(* CoDeSys 2.3.9.41 project: hlor-rezerv.pro *)
(* Libraries: STANDARD.LIB 4.10.05 11:14:46, IECSFC.LIB 13.4.06 15:51:28, ANALYZATION.LIB 5.10.99 09:05:06 *)

(* PLC configuration (modules and I/O channels)
Fast discrete inputs [I_SIMPLE_INPUT] node 0, in %IB0 out %QB0 {ChannellName = Fast discrete inputs; Filtrationtime = 10000}
  AT %IX0.0 [BitInput] Discrete input 1 {ChannellName = Enter name}
  AT %IX0.1 [BitInput] Discrete input 2 {ChannellName = Enter name}
  AT %IX0.2 [BitInput] Discrete input 3 {ChannellName = Enter name}
  AT %IX0.3 [BitInput] Discrete input 4 {ChannellName = Enter name}
Discrete inputs [ID130] node 1, in %IB1 out %QB1 {ChannellName = Discrete inputs; Filtrationtime_GeneralINP = 10; PinCount = 12; Visibility = No}
  AT %IB1.0 [ByteInput] 8 discrete inputs {ChannellName = Enter name}
  AT %IB1.1 [ByteInput] 4 discrete inputs {ChannellName = Enter name}
Fast discrete outputs [OWEN_ID570] node 2, in %IB2 out %QB2 {ChannellName = Fast discrete outputs; SafeValueBool = FALSE; SafeValueBool = FALSE; SafeValueBool = FALSE; SafeValueBool = FALSE; Visibility = No}
  SolNasos AT %QX2.0 [BitOutput] Fast discrete output 1 {ChannellName = Enter name}
  WaterNasos AT %QX2.1 [BitOutput] Fast discrete output 2 {ChannellName = Enter name}
  Klapan AT %QX2.2 [BitOutput] Fast discrete output 3 {ChannellName = Enter name}
  Elektroliz AT %QX2.3 [BitOutput] Fast discrete output 4 {ChannellName = Enter name}
Discrete outputs [ID131] node 3, in %IB3 out %QB3 {ChannellName = Discrete outputs; SafeValueByte = 0; Visibility = No}
  AT %QB3.0 [ByteOutput] 8 discrete outputs {ChannellName = Enter name}
  AT %QB3.1 [ByteOutput] 8 discrete outputs {ChannellName = Enter name}
D_Volume_Bak AT %IR4.0 [FloatInputP] Объем бака {ChannellName = Fast analog input; AIN_TYPE = 4-20 mA; Peak_Filtr = 200; Flt_Ch = Off; TauRC = 10; MinFV = 0; MaxFV = 150}
D_Konduktivnost AT %IR4.1 [FloatInputP] D_Konduktivnost {ChannellName = Fast analog input; AIN_TYPE = 4-20 mA; Peak_Filtr = 200; Flt_Ch = Off; TauRC = 10; MinFV = 0; MaxFV = 200}
D_Volt AT %IR4.2 [FloatInputP] Ток выпрямителя {ChannellName = Fast analog input; AIN_TYPE = 4-20 mA; Peak_Filtr = 200; Flt_Ch = Off; TauRC = 10; MinFV = 0; MaxFV = 80}
D_Amper AT %IR4.3 [FloatInputP] Напряжение выпрямителя {ChannellName = Fast analog input; AIN_TYPE = 4-20 mA; Peak_Filtr = 200; Flt_Ch = Off; TauRC = 10; MinFV = 0; MaxFV = 200}
DT_Water_Input AT %IR4.4 [FloatInputP] Температура воды на входе {ChannellName = Fast analog input; AIN_TYPE = 4-20 mA; Peak_Filtr = 200; Flt_Ch = Off; TauRC = 10; MinFV = 0; MaxFV = 100}
DT_Water_output AT %IR4.5 [FloatInputP] Температура воды на выходе {ChannellName = Fast analog input; AIN_TYPE = 4-20 mA; Peak_Filtr = 200; Flt_Ch = Off; TauRC = 10; MinFV = 0; MaxFV = 100}
AT %IR4.6 [FloatInputP] {ChannellName = Fast analog input; AIN_TYPE = 4-20 mA; Peak_Filtr = 200; Flt_Ch = Off; TauRC = 10; MinFV = 0; MaxFV = 100}
AT %IR4.7 [FloatInputP] You need to reboot PLC after change AI configuration! {ChannellName = Fast analog input; AIN_TYPE = 4-20 mA; Peak_Filtr = 200; Flt_Ch = Off; TauRC = 10; MinFV = 0; MaxFV = 20000.0}
AT %IW4.8 [WordInput] AI read time (10ms) {ChannellName = Enter name}
Analog outputs [ID126] node 5, in %IB5 out %QB5 {ChannellName = Analog outputs}
  AT %QR5.0 [FloatOutputP] AO #1 {ChannellName = Analog output; AOUT_TYPE = 4-20 mA; SafeValueREAL = 0.0}
  AT %QR5.1 [FloatOutputP] AO #2 {ChannellName = Analog output; AOUT_TYPE = 4-20 mA; SafeValueREAL = 0.0}
  AT %QR5.2 [FloatOutputP] AO #3 {ChannellName = Analog output; AOUT_TYPE = 4-20 mA; SafeValueREAL = 0.0}
  AT %QR5.3 [FloatOutputP] AO #4 {ChannellName = Analog output; AOUT_TYPE = 4-20 mA; SafeValueREAL = 0.0}
Special input [ID103] node 6, in %IB6 out %QB6 {ChannellName = Special input}
  AT %IX6.0 [BitInput] Special input {ChannellName = Enter name}
Special output [ID104] node 7, in %IB7 out %QB7 {ChannellName = Special output}
  AT %QX7.0 [BitOutput] Special output {ChannellName = Enter name}
Modbus [MODBUS_ID302] node 0, in %IB8.0 out %QB8.0 {ChannellName = Modbus}
  TCP [TCP_ID221] node 0, in %IB8.0.0 out %QB8.0.0 {ChannellName = TCP; RemotePort = 502; Visibility = No}
8 bits [8Bit] node 1, in %IB8.1 out %QB8.1 {ChannellName = 8 bit}
  AT %QB8.1.0 [ByteOutput] {ChannellName = Enter name}
8 bits [8Bit] node 2, in %IB8.2 out %QB8.2 {ChannellName = 8 bit}
  AT %QB8.2.0 [ByteOutput] {ChannellName = Enter name}
8 bits [8Bit] node 3, in %IB8.3 out %QB8.3 {ChannellName = 8 bit}
  AT %QB8.3.0 [ByteOutput] {ChannellName = Enter name}
8 bits [8Bit] node 4, in %IB8.4 out %QB8.4 {ChannellName = 8 bit}
  AT %QB8.4.0 [ByteOutput] {ChannellName = Enter name}
8 bits [8Bit] node 5, in %IB8.5 out %QB8.5 {ChannellName = 8 bit}
  AT %QB8.5.0 [ByteOutput] {ChannellName = Enter name}
8 bits [8Bit] node 6, in %IB8.6 out %QB8.6 {ChannellName = 8 bit}
  AT %QB8.6.0 [ByteOutput] {ChannellName = Enter name}
Float [Float] node 7, in %IB8.7 out %QB8.7 {ChannellName = float}
  D_Volume_Bak_SPK AT %QD8.7.0 [FloatOutput] {ChannellName = Enter name}
Float [Float] node 8, in %IB8.8 out %QB8.8 {ChannellName = float}
  D_Konduktivnost_SPK AT %QD8.8.0 [FloatOutput] {ChannellName = Enter name}
  D_Volt_SPK AT %QD8.9.0 [FloatOutput] {ChannellName = Enter name}
  D_Amper_SPK AT %QD8.10.0 [FloatOutput] {ChannellName = Enter name}
Float [Float] node 11, in %IB8.11 out %QB8.11 {ChannellName = float}
  DT_Water_Input_SPK AT %QD8.11.0 [FloatOutput] {ChannellName = Enter name}
Float [Float] node 12, in %IB8.12 out %QB8.12 {ChannellName = float}
  DT_Water_output_SPK AT %QD8.12.0 [FloatOutput] {ChannellName = Enter name}
8 bits [8Bit] node 13, in %IB8.13 out %QB8.13 {ChannellName = 8 bit}
  AT %QB8.13.0 [ByteOutput] {ChannellName = Enter name}
8 bits [8Bit] node 14, in %IB8.14 out %QB8.14 {ChannellName = 8 bit}
  AT %QB8.14.0 [ByteOutput] {ChannellName = Enter name}
8 bits [8Bit] node 15, in %IB8.15 out %QB8.15 {ChannellName = 8 bit}
  AT %QB8.15.0 [ByteOutput] {ChannellName = Enter name}
8 bits [8Bit] node 16, in %IB8.16 out %QB8.16 {ChannellName = 8 bit}
  AT %QB8.16.0 [ByteOutput] {ChannellName = Enter name}
*)

(* Task configuration *)
TASK NewTask (PRIORITY := 1, INTERVAL := T#200ms);
	PLC_PRG();
END_TASK

(* Global variable list: Global_Variables *)
VAR_GLOBAL
	PLAY_Elektroliz: BOOL;
	StartElectroliz: BOOL;
	StopElectroliz: BOOL;
	StartKlap: BOOL;
	StoptKlap: BOOL;
	StartWaterNasos: BOOL;
	StopWaterNasos: BOOL;
	StartSolNasos: BOOL;
	StopSolNasos: BOOL;
	StartHlorNasos1: BOOL;
	StopHlorNasos1: BOOL;
	StartHlorNasos2: BOOL;
	StopHlorNasos2: BOOL;

	StartVozduh: BOOL;
	StopVozduh: BOOL;
END_VAR

(* POU PLC_PRG, CFC *)
(*
	Программа управления гипохлоридной установкой
	Контроллер ОВЕН ПЛК-160 M2
	Панель оператора Kinko MT4404T

*)


PROGRAM PLC_PRG
VAR
	Electroliz_prg: Electroliz;
	Hlorirovanie_prg: Hlorirovanie;
	SoftWater_prg: SoftWater;
	SolNasos_prg: SolNasos;
	Vozduh_prg: Vozduh;
	D_Elektroliz_prg: D_Elektroliz;
END_VAR
VAR (* helpers for the ST form of the networks *)
	_t97 : WORD;
	_t98 : WORD;
	_t99 : WORD;
	_t100 : WORD;
	_t101 : WORD;
	_t204 : WORD;
END_VAR
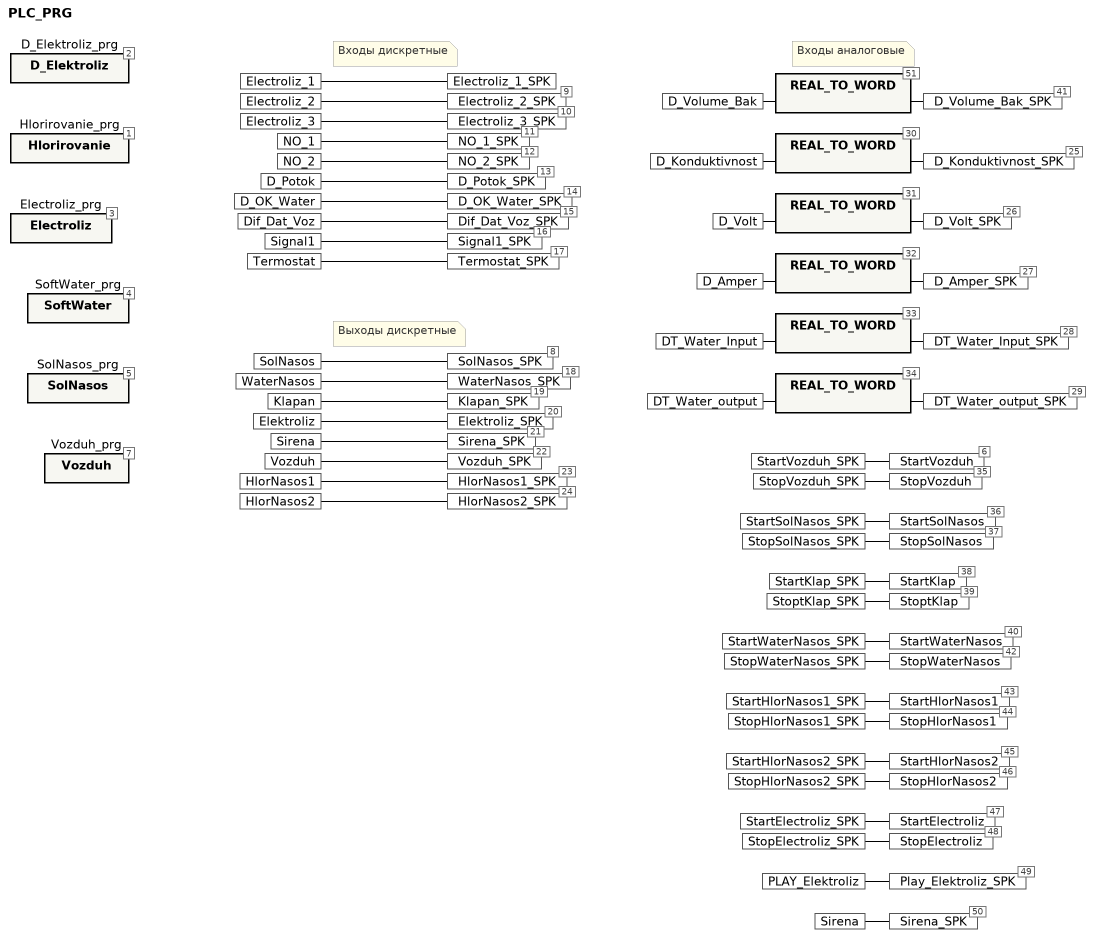
_CFC_ (* Continuous Function Chart, elements in execution order *)
#0 Electroliz_1_SPK <= Electroliz_1
#1 Hlorirovanie_prg:Hlorirovanie()
(* Входы дискретные *)
#2 D_Elektroliz_prg:D_Elektroliz()
#3 Electroliz_prg:Electroliz()
#4 SoftWater_prg:SoftWater()
#5 SolNasos_prg:SolNasos()
#6 StartVozduh <= StartVozduh_SPK
#7 Vozduh_prg:Vozduh()
(* Выходы дискретные *)
#8 SolNasos_SPK <= SolNasos
#9 Electroliz_2_SPK <= Electroliz_2
#10 Electroliz_3_SPK <= Electroliz_3
#11 NO_1_SPK <= NO_1
#12 NO_2_SPK <= NO_2
#13 D_Potok_SPK <= D_Potok
#14 D_OK_Water_SPK <= D_OK_Water
#15 Dif_Dat_Voz_SPK <= Dif_Dat_Voz
#16 Signal1_SPK <= Signal1
#17 Termostat_SPK <= Termostat
#18 WaterNasos_SPK <= WaterNasos
#19 Klapan_SPK <= Klapan
#20 Elektroliz_SPK <= Elektroliz
#21 Sirena_SPK <= Sirena
#22 Vozduh_SPK <= Vozduh
#23 HlorNasos1_SPK <= HlorNasos1
#24 HlorNasos2_SPK <= HlorNasos2
(* Входы аналоговые *)
#25 D_Konduktivnost_SPK <= #30
#26 D_Volt_SPK <= #31
#27 D_Amper_SPK <= #32
#28 DT_Water_Input_SPK <= #33
#29 DT_Water_output_SPK <= #34
#30 REAL_TO_WORD(D_Konduktivnost)
#31 REAL_TO_WORD(D_Volt)
#32 REAL_TO_WORD(D_Amper)
#33 REAL_TO_WORD(DT_Water_Input)
#34 REAL_TO_WORD(DT_Water_output)
#35 StopVozduh <= StopVozduh_SPK
#36 StartSolNasos <= StartSolNasos_SPK
#37 StopSolNasos <= StopSolNasos_SPK
#38 StartKlap <= StartKlap_SPK
#39 StoptKlap <= StoptKlap_SPK
#40 StartWaterNasos <= StartWaterNasos_SPK
#41 D_Volume_Bak_SPK <= #51
#42 StopWaterNasos <= StopWaterNasos_SPK
#43 StartHlorNasos1 <= StartHlorNasos1_SPK
#44 StopHlorNasos1 <= StopHlorNasos1_SPK
#45 StartHlorNasos2 <= StartHlorNasos2_SPK
#46 StopHlorNasos2 <= StopHlorNasos2_SPK
#47 StartElectroliz <= StartElectroliz_SPK
#48 StopElectroliz <= StopElectroliz_SPK
#49 Play_Elektroliz_SPK <= PLAY_Elektroliz
#50 Sirena_SPK <= Sirena
#51 REAL_TO_WORD(D_Volume_Bak)
_END_CFC_
(* the same logic as Structured Text *)
Electroliz_1_SPK := Electroliz_1;
Hlorirovanie_prg();
(* Входы дискретные *)
D_Elektroliz_prg();
Electroliz_prg();
SoftWater_prg();
SolNasos_prg();
StartVozduh := StartVozduh_SPK;
Vozduh_prg();
(* Выходы дискретные *)
SolNasos_SPK := SolNasos;
Electroliz_2_SPK := Electroliz_2;
Electroliz_3_SPK := Electroliz_3;
NO_1_SPK := NO_1;
NO_2_SPK := NO_2;
D_Potok_SPK := D_Potok;
D_OK_Water_SPK := D_OK_Water;
Dif_Dat_Voz_SPK := Dif_Dat_Voz;
Signal1_SPK := Signal1;
Termostat_SPK := Termostat;
WaterNasos_SPK := WaterNasos;
Klapan_SPK := Klapan;
Elektroliz_SPK := Elektroliz;
Sirena_SPK := Sirena;
Vozduh_SPK := Vozduh;
HlorNasos1_SPK := HlorNasos1;
HlorNasos2_SPK := HlorNasos2;
(* Входы аналоговые *)
D_Konduktivnost_SPK := _t97;
D_Volt_SPK := _t98;
D_Amper_SPK := _t99;
DT_Water_Input_SPK := _t100;
DT_Water_output_SPK := _t101;
_t97 := REAL_TO_WORD(D_Konduktivnost);
_t98 := REAL_TO_WORD(D_Volt);
_t99 := REAL_TO_WORD(D_Amper);
_t100 := REAL_TO_WORD(DT_Water_Input);
_t101 := REAL_TO_WORD(DT_Water_output);
StopVozduh := StopVozduh_SPK;
StartSolNasos := StartSolNasos_SPK;
StopSolNasos := StopSolNasos_SPK;
StartKlap := StartKlap_SPK;
StoptKlap := StoptKlap_SPK;
StartWaterNasos := StartWaterNasos_SPK;
D_Volume_Bak_SPK := _t204;
StopWaterNasos := StopWaterNasos_SPK;
StartHlorNasos1 := StartHlorNasos1_SPK;
StopHlorNasos1 := StopHlorNasos1_SPK;
StartHlorNasos2 := StartHlorNasos2_SPK;
StopHlorNasos2 := StopHlorNasos2_SPK;
StartElectroliz := StartElectroliz_SPK;
StopElectroliz := StopElectroliz_SPK;
Play_Elektroliz_SPK := PLAY_Elektroliz;
Sirena_SPK := Sirena;
_t204 := REAL_TO_WORD(D_Volume_Bak);
END_PROGRAM

(* POU Electroliz, CFC *)
(*
	Управление электролизером (выпрямитель)
	
	Кнопка StartElectroliz - включает электролизер. Кнопка активна только при включенном мягком насосе
	Кнопка StopElectroliz - выключает электролизер

	Датчик уровня солевого раствора
	При значениях <250 производит выключение электролизера с блокировкой кнопки включения электролизера
	При значениях >250 и состоянием "включено" - включает электролизер. Состояние запоминается исходя из ручных действий оператора

*)


FUNCTION_BLOCK Electroliz
VAR_INPUT
END_VAR
VAR_OUTPUT
END_VAR
VAR
	SR2: SR;
END_VAR
VAR (* helpers for the ST form of the networks *)
	_t25 : BOOL;
	_t50 : BOOL;
	_t14 : BOOL;
	_t29 : BOOL;
	_t31 : BOOL;
	_t52 : BOOL;
END_VAR
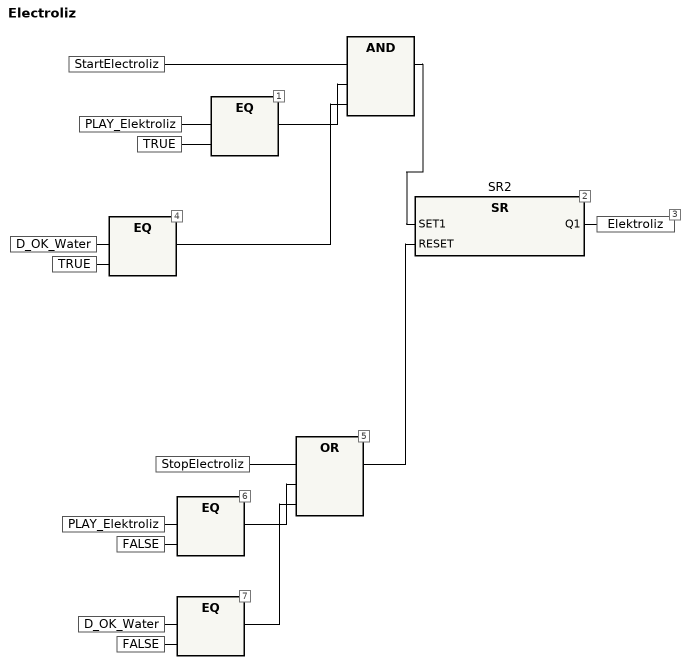
_CFC_ (* Continuous Function Chart, elements in execution order *)
#0 AND(StartElectroliz, #1, #4)
#1 EQ(PLAY_Elektroliz, TRUE)
#2 SR2:SR(SET1: #0, RESET: #5)
#3 Elektroliz <= #2.Q1
#4 EQ(D_OK_Water, TRUE)
#5 OR(StopElectroliz, #6, #7)
#6 EQ(PLAY_Elektroliz, FALSE)
#7 EQ(D_OK_Water, FALSE)
_END_CFC_
(* the same logic as Structured Text *)
_t14 := StartElectroliz AND _t25 AND _t50;
_t25 := PLAY_Elektroliz = TRUE;
SR2(SET1 := _t14, RESET := _t29);
Elektroliz := SR2.Q1;
_t50 := D_OK_Water = TRUE;
_t29 := StopElectroliz OR _t31 OR _t52;
_t31 := PLAY_Elektroliz = FALSE;
_t52 := D_OK_Water = FALSE;
END_FUNCTION_BLOCK

(* POU Hlorirovanie, CFC *)
(*
	Насосы первичного и вторичного хлорирования
	
	Насосы работют постоянно, независимо от других включенных/выключенных агрегатов
	Выключение насосов производится только в ручном режиме при отключении станции
	Без включенных насосов работа всех остальных агрегатов недопускается
	
	Кнопка StartHlorNasos1 - включает первичный насос хлорирования
	Кнопка StopHlorNasos1 - выключает первичный насос хлорирования
	Кнопка StartHlorNasos2 - включает вторичный насос хлорирования
	Кнопка StopHlorNasos2 - выключает вторичный насос хлорирования

	Датчик давления в баке выходного хлора. Установлен на дне бака
	Низкие значения датчика могут привести к полной остановке работы первичного и вторичного насосов

*)


FUNCTION_BLOCK Hlorirovanie
VAR_INPUT
END_VAR
VAR_OUTPUT
END_VAR
VAR
	SR3: SR;
	SR4: SR;
END_VAR
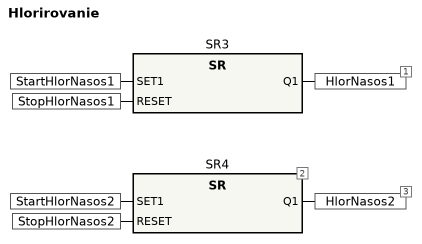
_CFC_ (* Continuous Function Chart, elements in execution order *)
#0 SR3:SR(SET1: StartHlorNasos1, RESET: StopHlorNasos1)
#1 HlorNasos1 <= #0.Q1
#2 SR4:SR(SET1: StartHlorNasos2, RESET: StopHlorNasos2)
#3 HlorNasos2 <= #2.Q1
_END_CFC_
(* the same logic as Structured Text *)
SR3(SET1 := StartHlorNasos1, RESET := StopHlorNasos1);
HlorNasos1 := SR3.Q1;
SR4(SET1 := StartHlorNasos2, RESET := StopHlorNasos2);
HlorNasos2 := SR4.Q1;
END_FUNCTION_BLOCK

(* POU SoftWater, CFC *)
(*
	Управление блоком мягкой воды

	Клапан:
	Кнопка StartKlap -  включение клапана. Кнопка активна только при включенном вентиляторе
	Кнопка StopKlap - выключение клапана. Кнопка активна только при выключенном насосе мягкой воды

	Насос:
	Кнопка StartWaterNasos - включение насоса мягкой воды. Кнопка активна только при включенном клапане
	Кнопка StopWaterNasos	- выключение насоса мягкой воды

*)





FUNCTION_BLOCK SoftWater
VAR_INPUT
END_VAR
VAR_OUTPUT
END_VAR
VAR
	SR6: SR;
	SR7: SR;
END_VAR
VAR (* helpers for the ST form of the networks *)
	_t25 : BOOL;
	_t24 : BOOL;
	_t32 : BOOL;
	_t40 : BOOL;
	_t43 : BOOL;
	_t47 : BOOL;
	_t48 : BOOL;
END_VAR
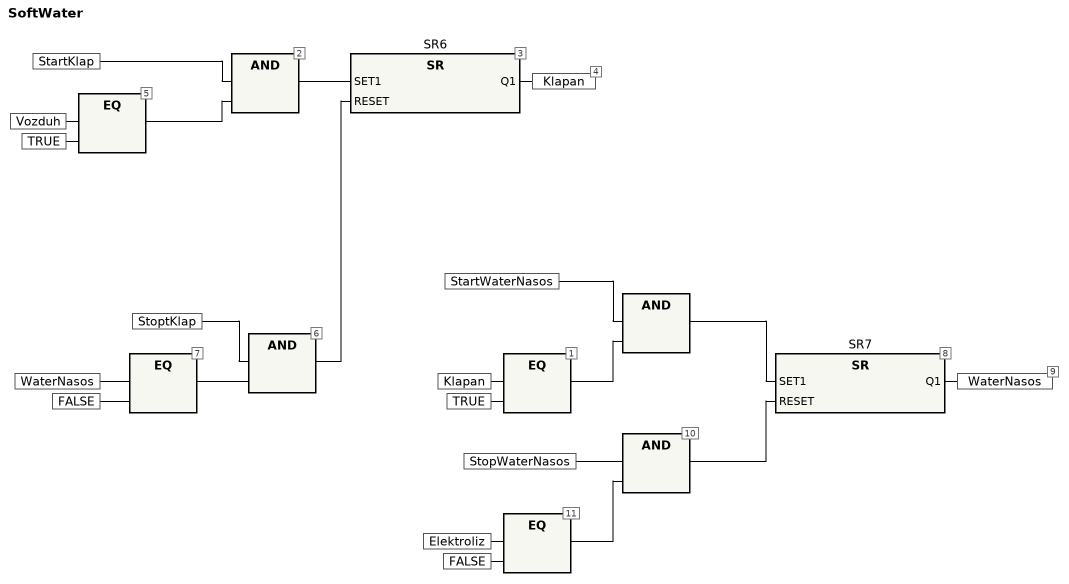
_CFC_ (* Continuous Function Chart, elements in execution order *)
#0 AND(StartWaterNasos, #1)
#1 EQ(Klapan, TRUE)
#2 AND(StartKlap, #5)
#3 SR6:SR(SET1: #2, RESET: #6)
#4 Klapan <= #3.Q1
#5 EQ(Vozduh, TRUE)
#6 AND(StoptKlap, #7)
#7 EQ(WaterNasos, FALSE)
#8 SR7:SR(SET1: #0, RESET: #10)
#9 WaterNasos <= #8.Q1
#10 AND(StopWaterNasos, #11)
#11 EQ(Elektroliz, FALSE)
_END_CFC_
(* the same logic as Structured Text *)
_t24 := StartWaterNasos AND _t25;
_t25 := Klapan = TRUE;
SR6(SET1 := StartKlap AND _t32, RESET := _t40);
Klapan := SR6.Q1;
_t32 := Vozduh = TRUE;
_t40 := StoptKlap AND _t43;
_t43 := WaterNasos = FALSE;
SR7(SET1 := _t24, RESET := _t47);
WaterNasos := SR7.Q1;
_t47 := StopWaterNasos AND _t48;
_t48 := Elektroliz = FALSE;
END_FUNCTION_BLOCK

(* POU Vozduh, CFC *)
(*
	Программа включения/выключения вентилятора

	Кнопка StartVoz - при нажатии запускает вентилятор и таймер 5 минут, после истечения времени таймера появляется возможность запуска следующих агрегатов
	Кнопка StopVoz - при нажатии запускает таймер 5 минут, после истечения времени таймера вентилятор выключается. Кнопка выключения заблокирована во время работы других систем

*)


FUNCTION_BLOCK Vozduh
VAR
	SR1: SR;

END_VAR
VAR_INPUT
END_VAR
VAR (* helpers for the ST form of the networks *)
	_t106 : BOOL;
	_t124 : BOOL;
	_t120 : BOOL;
END_VAR
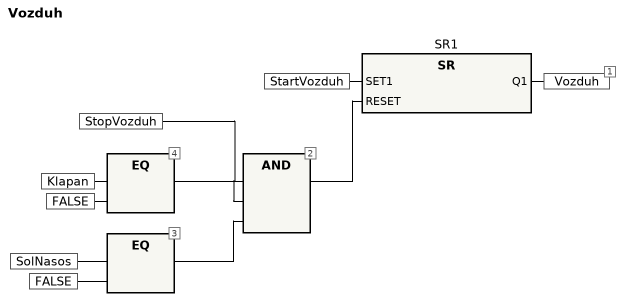
_CFC_ (* Continuous Function Chart, elements in execution order *)
#0 SR1:SR(SET1: StartVozduh, RESET: #2)
#1 Vozduh <= #0.Q1
#2 AND(StopVozduh, #4, #3)
#3 EQ(SolNasos, FALSE)
#4 EQ(Klapan, FALSE)
_END_CFC_
(* the same logic as Structured Text *)
SR1(SET1 := StartVozduh, RESET := _t106);
Vozduh := SR1.Q1;
_t106 := StopVozduh AND _t124 AND _t120;
_t120 := SolNasos = FALSE;
_t124 := Klapan = FALSE;
END_FUNCTION_BLOCK

(* POU SolNasos, CFC *)
(*
	Программа включения/выключения солевого насоса

	Кнопка StartSolNasos - производит включение солевого насоса
	Кнопка StopSolNasos - производит выключение солевого насоса

*)


FUNCTION_BLOCK SolNasos
VAR_INPUT
END_VAR
VAR_OUTPUT
END_VAR
VAR
	SR5: SR;
END_VAR
VAR (* helpers for the ST form of the networks *)
	_t26 : BOOL;
	_t27 : BOOL;
END_VAR
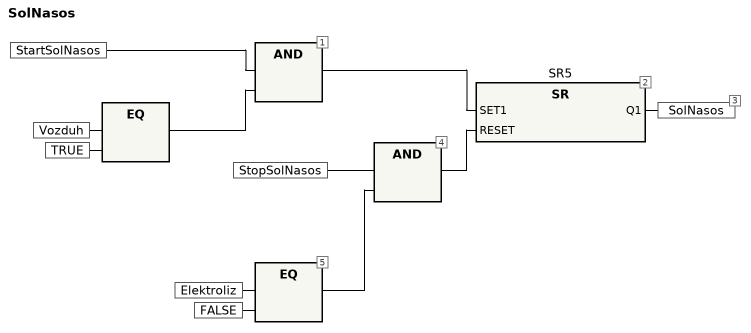
_CFC_ (* Continuous Function Chart, elements in execution order *)
#0 EQ(Vozduh, TRUE)
#1 AND(StartSolNasos, #0)
#2 SR5:SR(SET1: #1, RESET: #4)
#3 SolNasos <= #2.Q1
#4 AND(StopSolNasos, #5)
#5 EQ(Elektroliz, FALSE)
_END_CFC_
(* the same logic as Structured Text *)
SR5(SET1 := StartSolNasos AND (Vozduh = TRUE), RESET := _t26);
SolNasos := SR5.Q1;
_t26 := StopSolNasos AND _t27;
_t27 := Elektroliz = FALSE;
END_FUNCTION_BLOCK

(* POU D_Elektroliz, CFC *)
FUNCTION_BLOCK D_Elektroliz
VAR_INPUT
END_VAR
VAR_OUTPUT
END_VAR
VAR
	STOP_Elektroliz: BOOL;
	D_Volume_Bak1: REAL;
	DTWater: REAL;
	DTINPUTWATER: REAL;
END_VAR
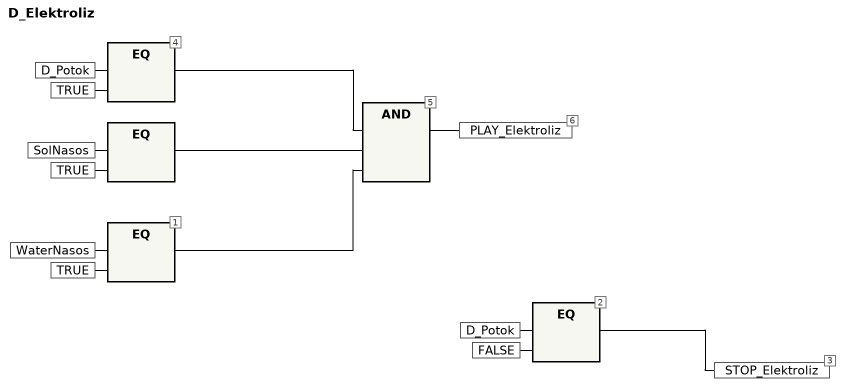
_CFC_ (* Continuous Function Chart, elements in execution order *)
#0 EQ(SolNasos, TRUE)
#1 EQ(WaterNasos, TRUE)
#2 EQ(D_Potok, FALSE)
#3 STOP_Elektroliz <= #2
#4 EQ(D_Potok, TRUE)
#5 AND(#4, #0, #1)
#6 PLAY_Elektroliz <= #5
_END_CFC_
(* the same logic as Structured Text *)
STOP_Elektroliz := D_Potok = FALSE;
PLAY_Elektroliz := (D_Potok = TRUE) AND (SolNasos = TRUE) AND (WaterNasos = TRUE);
END_FUNCTION_BLOCK

(* Visualisation Hlor
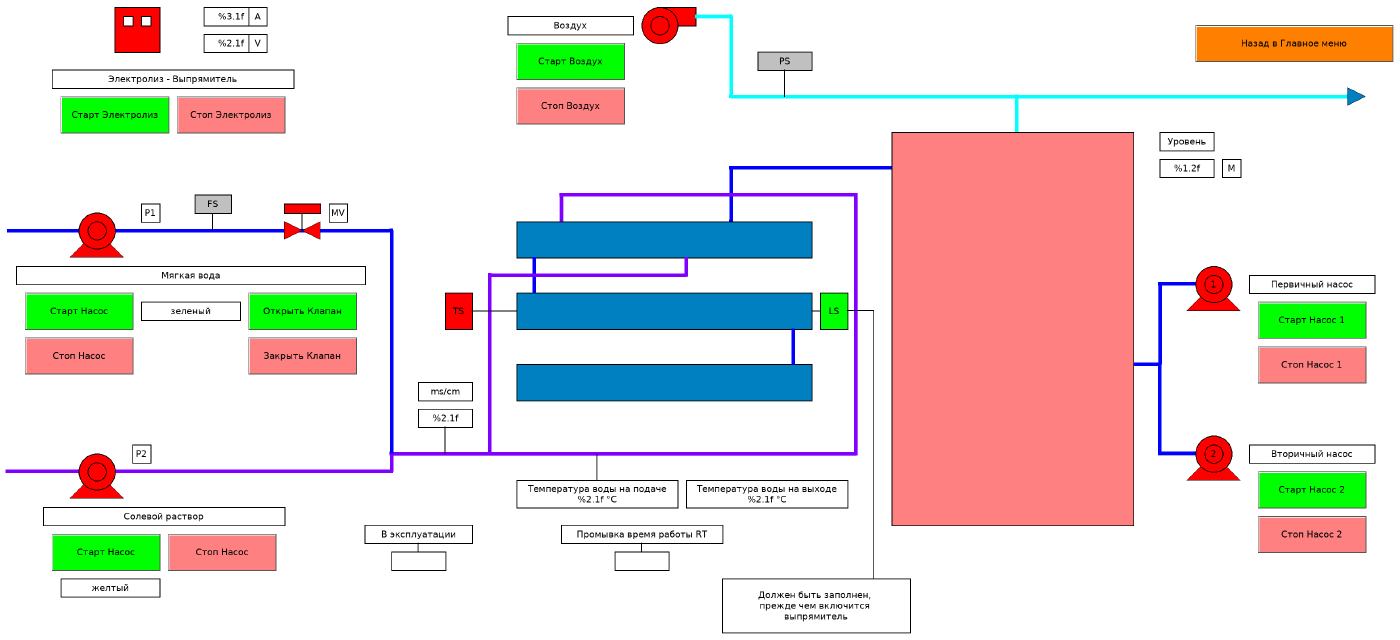
rectangle at (770,30)-(811,51): alarm colour if .Vozduh
button at (100,130)-(221,171): text "Старт Электролиз"; taps .StartElectroliz
button at (230,130)-(351,171): text "Стоп Электролиз"; taps .StopElectroliz
button at (610,70)-(731,111): text "Старт Воздух"; taps PLC_PRG.Vozduh_prg.StartVozduh
button at (610,120)-(731,161): text "Стоп Воздух"; taps PLC_PRG.Vozduh_prg.StopVozduh
button at (1370,50)-(1591,91): text "Назад в Главное меню"
button at (60,350)-(181,391): text "Старт Насос"; taps .StartWaterNasos
button at (60,400)-(181,441): text "Стоп Насос"; taps .StopWaterNasos
button at (310,350)-(431,391): text "Открыть Клапан"; taps .StartKlap
button at (310,400)-(431,441): text "Закрыть Клапан"; taps .StoptKlap
button at (1440,550)-(1561,591): text "Старт Насос 2"; taps .StartHlorNasos2
button at (1440,600)-(1561,641): text "Стоп Насос 2"; taps .StopHlorNasos2
button at (90,620)-(211,661): text "Старт Насос"; taps .StartSolNasos
button at (220,620)-(341,661): text "Стоп Насос"; taps .StopSolNasos
rectangle at (50,320)-(441,341): text "Мягкая вода"
rectangle at (90,100)-(361,121): text "Электролиз - Выпрямитель"
rectangle at (600,40)-(741,61): text "Воздух"
rectangle at (80,590)-(351,611): text "Солевой раствор"
rectangle at (1430,330)-(1571,351): text "Первичный насос"
rectangle at (1430,520)-(1571,541): text "Вторичный насос"
button at (1440,360)-(1561,401): text "Старт Насос 1"; taps .StartHlorNasos1
button at (1440,410)-(1561,451): text "Стоп Насос 1"; taps .StopHlorNasos1
rectangle at (160,30)-(211,81): alarm colour if .Electroliz
rounded rectangle at (260,30)-(321,51): text "%3.1f"; shows .D_Amper
rounded rectangle at (260,60)-(321,81): text "%2.1f"; shows .D_Volt
rounded rectangle at (880,80)-(941,101): text "PS"; alarm colour if .Vozduh
rounded rectangle at (1330,200)-(1391,221): text "%1.2f"; shows .D_Volume_Bak
rounded rectangle at (610,560)-(791,591): text "Температура воды на подаче / %2.1f °С"; shows .DT_Water_Input
rounded rectangle at (500,480)-(561,501): text "%2.1f"; shows .D_Konduktivnost
ellipse at (750,30)-(791,71): alarm colour if .Vozduh
polygon at (370,270)-(390,290): alarm colour if .Klapan
polygon at (350,270)-(370,290): alarm colour if .Klapan
rectangle at (350,250)-(391,261): alarm colour if .Klapan
rectangle at (250,240)-(291,261): text "FS"; alarm colour if .PLAY_Elektroliz
polygon at (110,280)-(170,310): alarm colour if .WaterNasos
ellipse at (120,260)-(161,301): alarm colour if .WaterNasos
ellipse at (130,270)-(151,291): alarm colour if .WaterNasos
polygon at (1360,340)-(1420,370): alarm colour if .HlorNasos1
ellipse at (1370,320)-(1411,361): alarm colour if .HlorNasos1
ellipse at (1380,330)-(1401,351): text "1"; alarm colour if .HlorNasos1
polygon at (1360,530)-(1420,560): alarm colour if .HlorNasos2
ellipse at (1370,510)-(1411,551): alarm colour if .HlorNasos2
ellipse at (1380,520)-(1401,541): text "2"; alarm colour if .HlorNasos2
ellipse at (760,40)-(781,61): alarm colour if .Vozduh
rectangle at (440,610)-(561,631): text "В эксплуатации"
rectangle at (660,610)-(841,631): text "Промывка время работы RT"
polygon at (110,550)-(170,580): alarm colour if .SolNasos
ellipse at (120,530)-(161,571): alarm colour if .SolNasos
ellipse at (130,540)-(151,561): alarm colour if .SolNasos
rectangle at (1330,170)-(1391,191): text "Уровень"
rounded rectangle at (310,30)-(331,51): text "A"
rounded rectangle at (310,60)-(331,81): text "V"
rounded rectangle at (950,350)-(981,391): text "LS"; alarm colour if .D_OK_Water
rounded rectangle at (530,350)-(561,391): text "TS"; alarm colour if .Termostat
rounded rectangle at (500,450)-(561,471): text "ms/cm"
rounded rectangle at (400,250)-(421,271): text "MV"
rounded rectangle at (1400,200)-(1421,221): text "M"
rounded rectangle at (190,250)-(211,271): text "P1"
rounded rectangle at (180,520)-(201,541): text "P2"
rectangle at (840,670)-(1051,731): text "Должен быть заполнен, / прежде чем включится / выпрямитель"
rounded rectangle at (800,560)-(981,591): text "Температура воды на выходе / %2.1f °С"; shows .DT_Water_output
rectangle at (100,670)-(211,691): text "желтый"
rectangle at (190,360)-(301,381): text "зеленый"
30 more shapes without text or variables
*)
